(* IEC 61131-3 sources: volt/packages/volt-lsp-iec/test-corpus/lenze-mid/Device/Plc Logic/Application/Library Manager/(unresolved)/iodriver parameter interfaces, 3 files *)

(* ---- INTERFACEIDS.gvl ---- *)
VAR_GLOBAL
	ITFID_ICMPIODRVPARAMETER : DWORD := 16#23;
END_VAR

(* ---- ICMPIODRVPARAMETER.itf ---- *)
INTERFACE ICMPIODRVPARAMETER
END_INTERFACE

METHOD IODRVREADPARAMETER : UDINT
VAR_INPUT
	PCONNECTOR : POINTER TO IoConfigConnector;
	PPARAMETER : POINTER TO IoConfigParameter;
	PDATA : POINTER TO BYTE;
	DWBITSIZE : DWORD;
	DWBITOFFSET : DWORD;
END_VAR
END_METHOD

METHOD IODRVWRITEPARAMETER : UDINT
VAR_INPUT
	PCONNECTOR : POINTER TO IoConfigConnector;
	PPARAMETER : POINTER TO IoConfigParameter;
	PDATA : POINTER TO BYTE;
	DWBITSIZE : DWORD;
	DWBITOFFSET : DWORD;
END_VAR
END_METHOD

(* ---- ICMPIODRVPARAMETER2.itf ---- *)
INTERFACE ICMPIODRVPARAMETER2
END_INTERFACE

METHOD IODRVREADPARAMETERBYID : UDINT
VAR_INPUT
	PCONNECTOR : POINTER TO IoConfigConnector;
	DWPARAMID : DWORD;
	PDATA : POINTER TO BYTE;
	DWBITSIZE : DWORD;
	DWBITOFFSET : DWORD;
END_VAR
END_METHOD

METHOD IODRVWRITEPARAMETERBYID : UDINT
VAR_INPUT
	PCONNECTOR : POINTER TO IoConfigConnector;
	DWPARAMID : DWORD;
	PDATA : POINTER TO BYTE;
	DWBITSIZE : DWORD;
	DWBITOFFSET : DWORD;
END_VAR
END_METHOD
